% RSLogix 500 project PID Temperature Control.RSS, saved by version 8.30.00.16 %
PROJECT "UNTITLED"    % processor: Bul.1763 MicroLogix 1100 Series B %

PROGRAM FILES
  LAD 2   9 rungs

DATA FILES
  O0 OUTPUT  9 elements
  I1 INPUT  16 elements
  S2 STATUS  66 elements
  B3 BINARY  1 elements
  T4 TIMER  1 elements
  C5 COUNTER  1 elements
  R6 CONTROL  1 elements
  N7 INTEGER  1 elements
  F8 FLOAT  1 elements
  PD9 TEMP  1 elements

LADDER 2
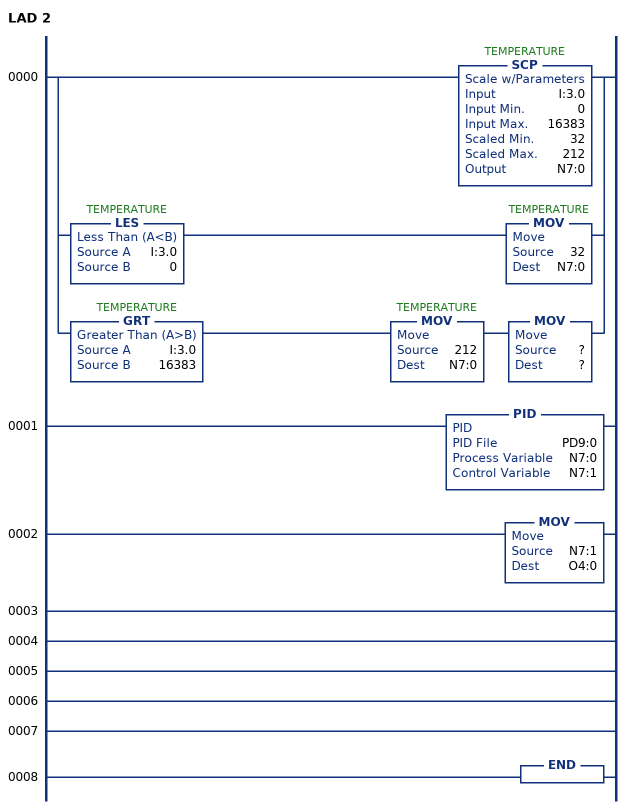
% Rung: 0 %  % edit flag set %
SOR BST SCP I:3.0 0 16383 32 212 N7:0 NXB LES I:3.0 0 MOV 32 N7:0 NXB GRT I:3.0 16383 MOV 212 N7:0 MOV ? ? BND EOR
%   I:3.0  "TEMPERATURE" %
%   N7:0  "TEMPERATURE" %
% Rung: 1 %  % edit flag set %
SOR PID PD9:0 N7:0 N7:1 EOR
%   N7:0  "TEMPERATURE" %
%   N7:1  "PID OUTPUT" %
% Rung: 2 %  % edit flag set %
SOR MOV N7:1 O4:0 EOR
%   N7:1  "PID OUTPUT" %
% Rung: 3 %  % edit flag set %
SOR EOR
% Rung: 4 %  % edit flag set %
SOR EOR
% Rung: 5 %  % edit flag set %
SOR EOR
% Rung: 6 %  % edit flag set %
SOR EOR
% Rung: 7 %  % edit flag set %
SOR EOR
% Rung: 8 %
SOR END EOR

OTHER DOCUMENTED ADDRESSES
  B3:0/0  "LOW TEMP SWITCH"
  B3:0/1  "HIGH SWITCH"
  B3:0/2  "HEATER"
  I:0  "TEMP SENSOR INPUT"
  I:1.0/0  "LOW TEMP SWITCH INPUT"
  I:1.0/1  "HIGH SWITCH INPUT"
  I:3.0/0  "TEMP SENSOR INPUT"
  O:0  "TEMP CONTROLLER"
  O:2.0/0  "HEATER OUTPUT"
